// TIA Portal V17 export
// export: Created 2022-07-16T16:56:12.9646662Z, ExportSetting WithDefaults, DisplayName Totally Integrated Automation Portal, DisplayVersion V17, DisplayName TIA Portal Openness, DisplayVersion V17, DisplayName TIA Portal Version Control Interface, DisplayVersion V17, DisplayName TIA Portal Test Suite Advanced, DisplayVersion V17, DisplayName STEP 7 Professional, DisplayVersion V17, DisplayName STEP 7 Safety, DisplayVersion V17, DisplayName WinCC Professional, DisplayVersion V17
TYPE "Client interface_1.dbData.postTestResult"
// stored: IsFailsafeCompliant false
   STRUCT
      preTestCheckSequence { ExternalWritable := 'False'; S7_SetPoint := 'True'} : "Client interface_1.dbData.postTestResult.preTestCheckSequence";
      mainSequence { ExternalWritable := 'False'; S7_SetPoint := 'True'} : "Client interface_1.dbData.postTestResult.mainSequence";
   END_STRUCT;
END_TYPE
